PROGRAM KL3208Comm
VAR
END_VAR

HWVar.KL3208Config(
	bConfigurate:= TRUE, 
	bReadConfig:= TRUE, 
	iSetSensorType:= 0, 
	tTimeout:= T#5S, 
	bBusy=> , 
	bError=> , 
	iErrorId=> , 
	iState=> , 
	iDataIn=> , 
	iTerminalType=> , 
	iSpecialType=> , 
	iFirmwareVersion=> , 
	sDescription=> , 
	sSensorType=> , 
	stInData:= HWVar.stKL3208_in, 
	stOutData:= HWVar.stKL3208_out);

END_PROGRAM

(* stored: Version 1.1.0.1, ProductVersion 3.1.4022.18
   POU KL3208Comm: Id {497885ca-2d47-44bb-bfa9-7980200d9189}, SpecialFunc None *)
